LIN {X 0,Y 133.124,Z 628.442,A -85,B 0,C 180,E1 30265.468,E2 30265.468} C_VEL
LIN {X 0,Y 133.768,Z 632.313,A -85,B 0,C 180,E1 30267.956,E2 30267.956} C_VEL
LIN {X 0,Y 124.95,Z 704.982,A -85,B 0,C 180,E1 30269.571,E2 30269.571} C_VEL
LIN {X 0,Y 121.16,Z 722.547,A -85,B 0,C 180,E1 30270.356,E2 30270.356} C_VEL
LIN {X 0,Y 115.982,Z 738.768,A -85,B 0,C 180,E1 30271.408,E2 30271.408} C_VEL
LIN {X 0,Y 109.441,Z 754.057,A -85,B 0,C 180,E1 30272.804,E2 30272.804} C_VEL
LIN {X 0,Y 101.053,Z 769.32,A -85,B 0,C 180,E1 30274.789,E2 30274.789} C_VEL
LIN {X 0,Y 91.388,Z 783.576,A -85,B 0,C 180,E1 30277.512,E2 30277.512} C_VEL
LIN {X 0,Y 80.997,Z 796.178,A -85,B 0,C 180,E1 30281.146,E2 30281.146} C_VEL
LIN {X 0,Y 69.646,Z 807.764,A -85,B 0,C 180,E1 30286.439,E2 30286.439} C_VEL
LIN {X 0,Y 58.196,Z 817.89,A -85,B 0,C 180,E1 30294.255,E2 30294.255} C_VEL
LIN {X 0,Y 47.458,Z 826.442,A -85,B 0,C 180,E1 30306.401,E2 30306.401} C_VEL
LIN {X 0,Y 39.232,Z 833.487,A -85,B 0,C 180,E1 30325.612,E2 30325.612} C_VEL
LIN {X 0,Y 36.606,Z 838.637,A -85,B 0,C 180,E1 30350.796,E2 30350.796} C_VEL
LIN {X 0,Y 40.825,Z 841.992,A -85,B 0,C 180,E1 30375.252,E2 30375.252} C_VEL
LIN {X 0,Y 51.196,Z 843.729,A -85,B 0,C 180,E1 30393.942,E2 30393.942} C_VEL
LIN {X 0,Y 64.117,Z 843.598,A -85,B 0,C 180,E1 30405.2,E2 30405.2} C_VEL
LIN {X 0,Y 78.941,Z 841.629,A -85,B 0,C 180,E1 30412.722,E2 30412.722} C_VEL
LIN {X 0,Y 94.061,Z 837.982,A -85,B 0,C 180,E1 30417.697,E2 30417.697} C_VEL
LIN {X 0,Y 109.006,Z 832.754,A -85,B 0,C 180,E1 30421.171,E2 30421.171} C_VEL
LIN {X 0,Y 120.172,Z 827.677,A -85,B 0,C 180,E1 30423.226,E2 30423.226} C_VEL
LIN {X 0,Y 103.476,Z 835.962,A -85,B 0,C 180,E1 30425.592,E2 30425.592} C_VEL
LIN {X 0,Y 87.073,Z 842.287,A -85,B 0,C 180,E1 30429.062,E2 30429.062} C_VEL
LIN {X 0,Y 70.028,Z 847.086,A -85,B 0,C 180,E1 30434.891,E2 30434.891} C_VEL
LIN {X 0,Y 53.982,Z 850.107,A -85,B 0,C 180,E1 30444.83,E2 30444.83} C_VEL
LIN {X 0,Y 41.414,Z 851.293,A -85,B 0,C 180,E1 30461.549,E2 30461.549} C_VEL
LIN {X 0,Y 34.954,Z 850.734,A -85,B 0,C 180,E1 30488.173,E2 30488.173} C_VEL
LIN {X 0,Y 35.789,Z 849.384,A -85,B 0,C 180,E1 30508.402,E2 30508.402} C_VEL
LIN {X 0,Y 35.133,Z 844.648,A -85,B 0,C 180,E1 30535.273,E2 30535.273} C_VEL
LIN {X 0,Y 41.425,Z 837.942,A -85,B 0,C 180,E1 30558.442,E2 30558.442} C_VEL
LIN {X 0,Y 51.599,Z 829.69,A -85,B 0,C 180,E1 30573.049,E2 30573.049} C_VEL
LIN {X 0,Y 63.089,Z 820.008,A -85,B 0,C 180,E1 30581.976,E2 30581.976} C_VEL
LIN {X 0,Y 74.753,Z 808.939,A -85,B 0,C 180,E1 30587.644,E2 30587.644} C_VEL
LIN {X 0,Y 85.236,Z 797.294,A -85,B 0,C 180,E1 30591.24,E2 30591.24} C_VEL
LIN {X 0,Y 89.458,Z 791.484,A -85,B 0,C 180,E1 30593.103,E2 30593.103} C_VEL
LIN {X 0,Y 97.246,Z 777.678,A -85,B 0,C 180,E1 30598.264,E2 30598.264} C_VEL
LIN {X 0,Y 100.826,Z 771.247,A -85,B 0,C 180,E1 30599.703,E2 30599.703} C_VEL
LIN {X 0,Y 101.927,Z 769.314,A -85,B 0,C 180,E1 30599.913,E2 30599.913} C_VEL
LIN {X 0,Y 110.001,Z 753.895,A -85,B 0,C 180,E1 30600.945,E2 30600.945} C_VEL
LIN {X 0,Y 116.535,Z 737.703,A -85,B 0,C 180,E1 30601.677,E2 30601.677} C_VEL
LIN {X 0,Y 121.533,Z 720.199,A -85,B 0,C 180,E1 30602.282,E2 30602.282} C_VEL
LIN {X 0,Y 124.74,Z 702.234,A -85,B 0,C 180,E1 30602.723,E2 30602.723} C_VEL
LIN {X 0,Y 132.684,Z 635.627,A -85,B 0,C 180,E1 30603.998,E2 30603.998} C_VEL
LIN {X 0,Y 131.939,Z 632.627,A -85,B 0,C 180,E1 30606.9,E2 30606.9} C_VEL
LIN {X 0,Y 131.38,Z 630.452,A -85,B 0,C 180,E1 30610.082,E2 30610.082} C_VEL
LIN {X 0,Y 131.027,Z 629.677,A -85,B 0,C 180,E1 30613.684,E2 30613.684} C_VEL
LIN {X 0,Y 130.967,Z 629.957,A -85,B 0,C 180,E1 30616.637,E2 30616.637} C_VEL
LIN {X 0,Y 131.177,Z 632.004,A -85,B 0,C 180,E1 30620.526,E2 30620.526} C_VEL
LIN {X 0,Y 131.68,Z 635.655,A -85,B 0,C 180,E1 30624.088,E2 30624.088} C_VEL
LIN {X 0,Y 131.749,Z 636.651,A -85,B 0,C 180,E1 30624.638,E2 30624.638} C_VEL
LIN {X 0,Y 123.152,Z 705.865,A -85,B 0,C 180,E1 30625.983,E2 30625.983} C_VEL
LIN {X 0,Y 119.235,Z 723.474,A -85,B 0,C 180,E1 30626.67,E2 30626.67} C_VEL
LIN {X 0,Y 113.925,Z 739.648,A -85,B 0,C 180,E1 30627.571,E2 30627.571} C_VEL
LIN {X 0,Y 107.211,Z 754.907,A -85,B 0,C 180,E1 30628.757,E2 30628.757} C_VEL
LIN {X 0,Y 98.58,Z 770.166,A -85,B 0,C 180,E1 30630.442,E2 30630.442} C_VEL
LIN {X 0,Y 88.846,Z 784.086,A -85,B 0,C 180,E1 30632.698,E2 30632.698} C_VEL
LIN {X 0,Y 78.696,Z 796.083,A -85,B 0,C 180,E1 30635.594,E2 30635.594} C_VEL
LIN {X 0,Y 66.698,Z 807.856,A -85,B 0,C 180,E1 30640.132,E2 30640.132} C_VEL
LIN {X 0,Y 54.319,Z 818.147,A -85,B 0,C 180,E1 30647.07,E2 30647.07} C_VEL
LIN {X 0,Y 42.982,Z 826.417,A -85,B 0,C 180,E1 30657.651,E2 30657.651} C_VEL
LIN {X 0,Y 33.253,Z 833.324,A -85,B 0,C 180,E1 30676.078,E2 30676.078} C_VEL
LIN {X 0,Y 28.617,Z 838.842,A -85,B 0,C 180,E1 30706.228,E2 30706.228} C_VEL
LIN {X 0,Y 32.757,Z 842.681,A -85,B 0,C 180,E1 30737.811,E2 30737.811} C_VEL
LIN {X 0,Y 43.969,Z 844.72,A -85,B 0,C 180,E1 30758.797,E2 30758.797} C_VEL
LIN {X 0,Y 58.756,Z 844.922,A -85,B 0,C 180,E1 30770.741,E2 30770.741} C_VEL
LIN {X 0,Y 74.674,Z 843.253,A -85,B 0,C 180,E1 30777.696,E2 30777.696} C_VEL
LIN {X 0,Y 91.051,Z 839.669,A -85,B 0,C 180,E1 30782.179,E2 30782.179} C_VEL
LIN {X 0,Y 92.633,Z 839.232,A -85,B 0,C 180,E1 30782.524,E2 30782.524} C_VEL
LIN {X 0,Y 74.45,Z 844.692,A -85,B 0,C 180,E1 30786.387,E2 30786.387} C_VEL
LIN {X 0,Y 57.405,Z 848.129,A -85,B 0,C 180,E1 30792.746,E2 30792.746} C_VEL
LIN {X 0,Y 40.983,Z 849.825,A -85,B 0,C 180,E1 30805.492,E2 30805.492} C_VEL
LIN {X 0,Y 28.985,Z 849.655,A -85,B 0,C 180,E1 30832.499,E2 30832.499} C_VEL
LIN {X 0,Y 27.639,Z 847.886,A -85,B 0,C 180,E1 30867.931,E2 30867.931} C_VEL
LIN {X 0,Y 27.922,Z 842.961,A -85,B 0,C 180,E1 30902.494,E2 30902.494} C_VEL
LIN {X 0,Y 36.477,Z 836.037,A -85,B 0,C 180,E1 30928.187,E2 30928.187} C_VEL
LIN {X 0,Y 48.795,Z 827.319,A -85,B 0,C 180,E1 30942.102,E2 30942.102} C_VEL
LIN {X 0,Y 61.038,Z 817.679,A -85,B 0,C 180,E1 30949.383,E2 30949.383} C_VEL
LIN {X 0,Y 73.401,Z 806.264,A -85,B 0,C 180,E1 30953.947,E2 30953.947} C_VEL
LIN {X 0,Y 85.602,Z 792.771,A -85,B 0,C 180,E1 30957.065,E2 30957.065} C_VEL
LIN {X 0,Y 96.003,Z 778.816,A -85,B 0,C 180,E1 30959.013,E2 30959.013} C_VEL
LIN {X 0,Y 101.927,Z 769.314,A -85,B 0,C 180,E1 30959.913,E2 30959.913} C_VEL
LIN {X 0,Y 105.388,Z 762.627,A -85,B 0,C 180,E1 30960.932,E2 30960.932} C_VEL
LIN {X 0,Y 111.802,Z 746.124,A -85,B 0,C 180,E1 30964.626,E2 30964.626} C_VEL
LIN {X 0,Y 114.332,Z 738.962,A -85,B 0,C 180,E1 30965.495,E2 30965.495} C_VEL
LIN {X 0,Y 114.714,Z 737.92,A -85,B 0,C 180,E1 30965.539,E2 30965.539} C_VEL
LIN {X 0,Y 119.827,Z 720.664,A -85,B 0,C 180,E1 30965.992,E2 30965.992} C_VEL
LIN {X 0,Y 123.226,Z 702.456,A -85,B 0,C 180,E1 30966.353,E2 30966.353} C_VEL
LIN {X 0,Y 130.791,Z 640.674,A -85,B 0,C 180,E1 30967.309,E2 30967.309} C_VEL
LIN {X 0,Y 130.276,Z 638.224,A -85,B 0,C 180,E1 30970.764,E2 30970.764} C_VEL
LIN {X 0,Y 129.996,Z 637.59,A -85,B 0,C 180,E1 30974.705,E2 30974.705} C_VEL
LIN {X 0,Y 129.947,Z 638.429,A -85,B 0,C 180,E1 30977.463,E2 30977.463} C_VEL
LIN {X 0,Y 130.044,Z 639.857,A -85,B 0,C 180,E1 30979.774,E2 30979.774} C_VEL
LIN {X 0,Y 130.134,Z 641.399,A -85,B 0,C 180,E1 30981.234,E2 30981.234} C_VEL
LIN {X 0,Y 121.85,Z 706.742,A -85,B 0,C 180,E1 30982.302,E2 30982.302} C_VEL
LIN {X 0,Y 117.817,Z 724.395,A -85,B 0,C 180,E1 30982.878,E2 30982.878} C_VEL
LIN {X 0,Y 112.256,Z 740.896,A -85,B 0,C 180,E1 30983.63,E2 30983.63} C_VEL
LIN {X 0,Y 105.045,Z 756.675,A -85,B 0,C 180,E1 30984.629,E2 30984.629} C_VEL
LIN {X 0,Y 95.722,Z 772.527,A -85,B 0,C 180,E1 30986.061,E2 30986.061} C_VEL
LIN {X 0,Y 85.94,Z 785.915,A -85,B 0,C 180,E1 30987.842,E2 30987.842} C_VEL
LIN {X 0,Y 74.259,Z 798.903,A -85,B 0,C 180,E1 30990.487,E2 30990.487} C_VEL
LIN {X 0,Y 61.763,Z 810.377,A -85,B 0,C 180,E1 30994.345,E2 30994.345} C_VEL
LIN {X 0,Y 48.652,Z 820.401,A -85,B 0,C 180,E1 31000.498,E2 31000.498} C_VEL
LIN {X 0,Y 35.477,Z 828.887,A -85,B 0,C 180,E1 31011.678,E2 31011.678} C_VEL
LIN {X 0,Y 24.188,Z 835.906,A -85,B 0,C 180,E1 31035.635,E2 31035.635} C_VEL
LIN {X 0,Y 21.009,Z 841.031,A -85,B 0,C 180,E1 31078.414,E2 31078.414} C_VEL
LIN {X 0,Y 29.043,Z 844.39,A -85,B 0,C 180,E1 31113.512,E2 31113.512} C_VEL
LIN {X 0,Y 43.511,Z 846.133,A -85,B 0,C 180,E1 31131.144,E2 31131.144} C_VEL
LIN {X 0,Y 58.993,Z 846.026,A -85,B 0,C 180,E1 31139.403,E2 31139.403} C_VEL
LIN {X 0,Y 65.658,Z 845.494,A -85,B 0,C 180,E1 31141.813,E2 31141.813} C_VEL
LIN {X 0,Y 47.477,Z 847.981,A -85,B 0,C 180,E1 31148.204,E2 31148.204} C_VEL
LIN {X 0,Y 30.208,Z 848.67,A -85,B 0,C 180,E1 31163.399,E2 31163.399} C_VEL
LIN {X 0,Y 19.499,Z 847.492,A -85,B 0,C 180,E1 31202.523,E2 31202.523} C_VEL
LIN {X 0,Y 19.475,Z 846.366,A -85,B 0,C 180,E1 31227.062,E2 31227.062} C_VEL
LIN {X 0,Y 21.444,Z 841.228,A -85,B 0,C 180,E1 31274.386,E2 31274.386} C_VEL
LIN {X 0,Y 32.883,Z 834.132,A -85,B 0,C 180,E1 31300.503,E2 31300.503} C_VEL
LIN {X 0,Y 46.502,Z 825.476,A -85,B 0,C 180,E1 31311.538,E2 31311.538} C_VEL
LIN {X 0,Y 60.067,Z 815.218,A -85,B 0,C 180,E1 31317.159,E2 31317.159} C_VEL
LIN {X 0,Y 72.994,Z 803.496,A -85,B 0,C 180,E1 31320.417,E2 31320.417} C_VEL
LIN {X 0,Y 85.072,Z 790.211,A -85,B 0,C 180,E1 31322.524,E2 31322.524} C_VEL
LIN {X 0,Y 95.707,Z 775.754,A -85,B 0,C 180,E1 31323.869,E2 31323.869} C_VEL
LIN {X 0,Y 104.948,Z 760.149,A -85,B 0,C 180,E1 31324.773,E2 31324.773} C_VEL
LIN {X 0,Y 111.97,Z 745.106,A -85,B 0,C 180,E1 31325.327,E2 31325.327} C_VEL
LIN {X 0,Y 114.714,Z 737.92,A -85,B 0,C 180,E1 31325.539,E2 31325.539} C_VEL
LIN {X 0,Y 117.028,Z 730.64,A -85,B 0,C 180,E1 31326.224,E2 31326.224} C_VEL
LIN {X 0,Y 119.925,Z 717.271,A -85,B 0,C 180,E1 31328.633,E2 31328.633} C_VEL
LIN {X 0,Y 121.31,Z 708.786,A -85,B 0,C 180,E1 31329.803,E2 31329.803} C_VEL
LIN {X 0,Y 121.964,Z 704.408,A -85,B 0,C 180,E1 31330.034,E2 31330.034} C_VEL
LIN {X 0,Y 129.244,Z 646.329,A -85,B 0,C 180,E1 31330.809,E2 31330.809} C_VEL
LIN {X 0,Y 129.039,Z 645.563,A -85,B 0,C 180,E1 31333.443,E2 31333.443} C_VEL
LIN {X 0,Y 128.947,Z 645.834,A -85,B 0,C 180,E1 31335.948,E2 31335.948} C_VEL
LIN {X 0,Y 128.905,Z 646.885,A -85,B 0,C 180,E1 31337.764,E2 31337.764} C_VEL
LIN {X 0,Y 121.061,Z 707.617,A -85,B 0,C 180,E1 31338.557,E2 31338.557} C_VEL
LIN {X 0,Y 116.896,Z 725.43,A -85,B 0,C 180,E1 31339.015,E2 31339.015} C_VEL
LIN {X 0,Y 111.418,Z 741.399,A -85,B 0,C 180,E1 31339.561,E2 31339.561} C_VEL
LIN {X 0,Y 104.445,Z 756.602,A -85,B 0,C 180,E1 31340.252,E2 31340.252} C_VEL
LIN {X 0,Y 95.454,Z 771.863,A -85,B 0,C 180,E1 31341.207,E2 31341.207} C_VEL
LIN {X 0,Y 84.964,Z 786.147,A -85,B 0,C 180,E1 31342.51,E2 31342.51} C_VEL
LIN {X 0,Y 73.478,Z 798.817,A -85,B 0,C 180,E1 31344.254,E2 31344.254} C_VEL
LIN {X 0,Y 60.534,Z 810.47,A -85,B 0,C 180,E1 31346.878,E2 31346.878} C_VEL
LIN {X 0,Y 46.715,Z 820.679,A -85,B 0,C 180,E1 31351.11,E2 31351.11} C_VEL
LIN {X 0,Y 33.207,Z 828.869,A -85,B 0,C 180,E1 31358.473,E2 31358.473} C_VEL
LIN {X 0,Y 19.909,Z 835.738,A -85,B 0,C 180,E1 31376.459,E2 31376.459} C_VEL
LIN {X 0,Y 12.763,Z 841.239,A -85,B 0,C 180,E1 31433.052,E2 31433.052} C_VEL
LIN {X 0,Y 21.924,Z 845.018,A -85,B 0,C 180,E1 31483.266,E2 31483.266} C_VEL
LIN {X 0,Y 36.996,Z 847.06,A -85,B 0,C 180,E1 31499.249,E2 31499.249} C_VEL
LIN {X 0,Y 39.497,Z 847.231,A -85,B 0,C 180,E1 31500.824,E2 31500.824} C_VEL
LIN {X 0,Y 21.76,Z 847.068,A -85,B 0,C 180,E1 31515.239,E2 31515.239} C_VEL
LIN {X 0,Y 11.33,Z 845.135,A -85,B 0,C 180,E1 31576.071,E2 31576.071} C_VEL
LIN {X 0,Y 11.319,Z 844.786,A -85,B 0,C 180,E1 31584.941,E2 31584.941} C_VEL
LIN {X 0,Y 16.867,Z 839.341,A -85,B 0,C 180,E1 31655.491,E2 31655.491} C_VEL
LIN {X 0,Y 31.116,Z 832.192,A -85,B 0,C 180,E1 31674.991,E2 31674.991} C_VEL
LIN {X 0,Y 45.01,Z 823.915,A -85,B 0,C 180,E1 31681.466,E2 31681.466} C_VEL
LIN {X 0,Y 59.206,Z 813.546,A -85,B 0,C 180,E1 31684.86,E2 31684.86} C_VEL
LIN {X 0,Y 72.496,Z 801.692,A -85,B 0,C 180,E1 31686.76,E2 31686.76} C_VEL
LIN {X 0,Y 84.293,Z 788.798,A -85,B 0,C 180,E1 31687.915,E2 31687.915} C_VEL
LIN {X 0,Y 95.073,Z 774.236,A -85,B 0,C 180,E1 31688.662,E2 31688.662} C_VEL
LIN {X 0,Y 104.312,Z 758.667,A -85,B 0,C 180,E1 31689.139,E2 31689.139} C_VEL
LIN {X 0,Y 111.748,Z 742.442,A -85,B 0,C 180,E1 31689.434,E2 31689.434} C_VEL
LIN {X 0,Y 117.645,Z 724.841,A -85,B 0,C 180,E1 31689.732,E2 31689.732} C_VEL
LIN {X 0,Y 121.547,Z 707.248,A -85,B 0,C 180,E1 31689.997,E2 31689.997} C_VEL
LIN {X 0,Y 121.964,Z 704.408,A -85,B 0,C 180,E1 31690.034,E2 31690.034} C_VEL
LIN {X 0,Y 122.942,Z 696.798,A -85,B 0,C 180,E1 31690.605,E2 31690.605} C_VEL
LIN {X 0,Y 125.11,Z 676.745,A -85,B 0,C 180,E1 31693.697,E2 31693.697} C_VEL
LIN {X 0,Y 125.904,Z 670.191,A -85,B 0,C 180,E1 31694.082,E2 31694.082} C_VEL
LIN {X 0,Y 127.984,Z 653.633,A -85,B 0,C 180,E1 31694.248,E2 31694.248} C_VEL
LIN {X 0,Y 120.795,Z 708.466,A -85,B 0,C 180,E1 31694.78,E2 31694.78} C_VEL
LIN {X 0,Y 116.522,Z 726.42,A -85,B 0,C 180,E1 31695.108,E2 31695.108} C_VEL
LIN {X 0,Y 111.003,Z 742.263,A -85,B 0,C 180,E1 31695.46,E2 31695.46} C_VEL
LIN {X 0,Y 103.578,Z 758.123,A -85,B 0,C 180,E1 31695.899,E2 31695.899} C_VEL
LIN {X 0,Y 94.354,Z 773.452,A -85,B 0,C 180,E1 31696.455,E2 31696.455} C_VEL
LIN {X 0,Y 83.724,Z 787.613,A -85,B 0,C 180,E1 31697.175,E2 31697.175} C_VEL
LIN {X 0,Y 71.545,Z 800.642,A -85,B 0,C 180,E1 31698.133,E2 31698.133} C_VEL
LIN {X 0,Y 58.329,Z 812.156,A -85,B 0,C 180,E1 31699.47,E2 31699.47} C_VEL
LIN {X 0,Y 44.08,Z 822.248,A -85,B 0,C 180,E1 31701.559,E2 31701.559} C_VEL
LIN {X 0,Y 28.82,Z 830.81,A -85,B 0,C 180,E1 31705.566,E2 31705.566} C_VEL
LIN {X 0,Y 12.737,Z 837.937,A -85,B 0,C 180,E1 31718.914,E2 31718.914} C_VEL
LIN {X 0,Y 6.855,Z 843.195,A -85,B 0,C 180,E1 31834.033,E2 31834.033} C_VEL
LIN {X 0,Y 13.657,Z 845.051,A -85,B 0,C 180,E1 31858.657,E2 31858.657} C_VEL
LIN {X 0,Y 3.549,Z 843.335,A -85,B 0,C 180,E1 31925.033,E2 31925.033} C_VEL
LIN {X 0,Y 15.044,Z 837.714,A -85,B 0,C 180,E1 32044.385,E2 32044.385} C_VEL
LIN {X 0,Y 30.456,Z 830.739,A -85,B 0,C 180,E1 32049.958,E2 32049.958} C_VEL
LIN {X 0,Y 45.973,Z 821.66,A -85,B 0,C 180,E1 32051.834,E2 32051.834} C_VEL
LIN {X 0,Y 60.47,Z 811.048,A -85,B 0,C 180,E1 32052.687,E2 32052.687} C_VEL
LIN {X 0,Y 73.618,Z 799.148,A -85,B 0,C 180,E1 32053.131,E2 32053.131} C_VEL
LIN {X 0,Y 85.303,Z 786.098,A -85,B 0,C 180,E1 32053.373,E2 32053.373} C_VEL
LIN {X 0,Y 96.143,Z 771.171,A -85,B 0,C 180,E1 32053.494,E2 32053.494} C_VEL
LIN {X 0,Y 104.899,Z 755.945,A -85,B 0,C 180,E1 32053.531,E2 32053.531} C_VEL
LIN {X 0,Y 112.361,Z 739.068,A -85,B 0,C 180,E1 32053.543,E2 32053.543} C_VEL
LIN {X 0,Y 117.87,Z 721.987,A -85,B 0,C 180,E1 32053.65,E2 32053.65} C_VEL
LIN {X 0,Y 121.511,Z 704.333,A -85,B 0,C 180,E1 32053.795,E2 32053.795} C_VEL
LIN {X 0,Y 125.904,Z 670.191,A -85,B 0,C 180,E1 32054.082,E2 32054.082} C_VEL
LIN {X 0,Y 129.868,Z 670.442,A -85,B 0,C 180,E1 32054.261,E2 32054.261} C_VEL
LIN {X 0,Y 129.868,Z 931,A -85,B 0,C 180,E1 32054.261,E2 32054.261} C_VEL
LIN {X 0,Y 129.868,Z 931,A -85,B 0,C 180,E1 32054.261,E2 32054.261}

QRS_NEXT_CUT()

QRS_NEXT()
QRS_HOME()

END
